(* Schneider Machine Expert - Basic project first try step counter, file version 2.7.0.0 *)
(* ProjectInformations: Name=New project *)

HARDWARE
  Cpu 0: TM221M16R/G
  EthernetConfiguration: NetworkName=M221, IpAllocationMode=FixedAddress, IpAddress=0.0.0.0, SubnetMask=0.0.0.0
  SerialLineConfiguration: Baud=Baud19200, Parity=ParityEven, DataBits=DataBits8, StopBits=StopBits1, PhysicalMedium=PhysicalMediumRs485, TransmissionMode=TransmissionModeModbusRtu, SlaveId=1, Addressing=SlaveAddressing
  MastTask: UsePeriodScanMode=false, PeriodScan=100
  FastTask: Period=255
  CpuBehavior: StartingMode=StartAsPreviousState, AutoSaveRamOnEeprom=true, WatchdogPeriod=250

SYMBOLS  (address, symbol, comment, settings)
  %M0       RESET
  %M1       COUNT_UP
  %M2       COUNT_DOWN
  %SC0      STEP_COUNTER_0

POU New POU
  (* SectionNumber=1 *)

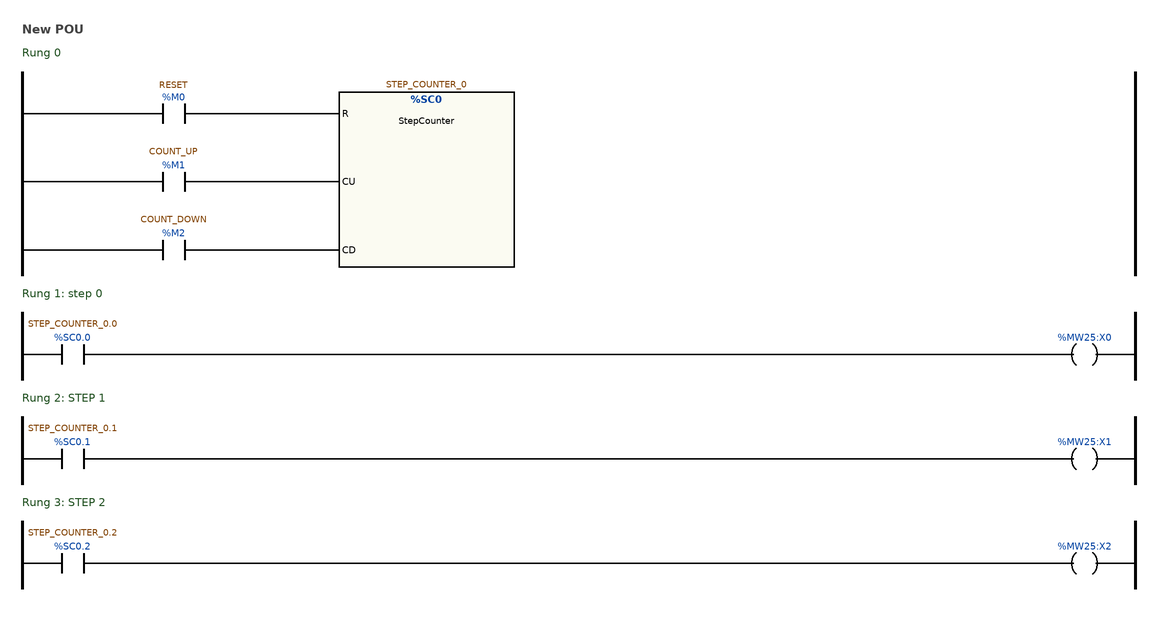

// Rung 0
  BLK %SC0                (* STEP_COUNTER_0 *)
  LD %M0                  (* RESET *)
  R
  LD %M1                  (* COUNT_UP *)
  CU
  LD %M2                  (* COUNT_DOWN *)
  CD
  END_BLK
  // as ST:
  //   STEP_COUNTER_0(R := RESET, CU := COUNT_UP, CD := COUNT_DOWN);

// Rung 1: step 0
  LD %SC0.0
  ST %MW25:X0
  // as ST:
  //   %MW25:X0 := %SC0.0;

// Rung 2: STEP 1
  LD %SC0.1
  ST %MW25:X1
  // as ST:
  //   %MW25:X1 := %SC0.1;

// Rung 3: STEP 2
  LD %SC0.2
  ST %MW25:X2
  // as ST:
  //   %MW25:X2 := %SC0.2;
